PROGRAM MAIN
VAR

	Axis		: AxisControl;
	State		: BYTE;
	
	Test		: AxisStates;
	

END_VAR


// Implement AxisControl

Axis.CyclicUpdate();

Axis.AutoErrorCheckAndReset();

Test := Axis.AxisStates;

CASE State OF
	
	0:
	
		IF Axis.PowerOn() THEN
			State := 1;
		END_IF
		
	1:
		IF Axis.WriteToParameter(Parameter := MC_AxisParameter.EnableLimitNeg, Value := 1) THEN
			State := 22;
		ELSE
			State := 55;
		END_IF
END_CASE

END_PROGRAM

(* stored: Version 1.1.0.1, ProductVersion 3.1.4024.12
   POU MAIN: Id {bdf002b2-15de-401c-9ee1-0af059a6100a}, SpecialFunc None *)
